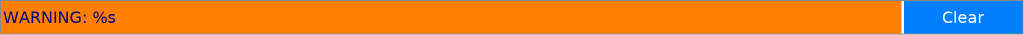
VISUALIZATION N_Footer_Alarm  // 1024x35
    Rectangle (0,0 902x35), "WARNING: %s", text variable: stWarningTxt1, invisible if: not bWrn2, input disabled if: not bWrn2
    Rectangle (0,0 902x35), "WARNING: %s", text variable: stWarningTxt, invisible if: not bWrn, input disabled if: not bWrn
    Rectangle (903,0 120x35), "Clear", invisible if: not bxoa, input disabled if: not bxoa
        OnMouseDown: execute {
            bWrn := FALSE;
            bWrn2 := FALSE;
            bWarning := FALSE;
            bWarning2 := FALSE;
            bxoa := FALSE;
            bSirens := false;
        }
END_VISUALIZATION

(* stored: Version 1.1.0.1, ProductVersion 3.1.4024.12
   Visu N_Footer_Alarm: Id {a59cfe85-a008-46f3-aaff-0cba6cf89eac} *)
